{attribute 'qualified_only'}
{attribute 'strict'}
TYPE Motor :
(
	RotationMotor := 0,
	LiftingMotor := 1,
	ExtensionMotor := 2,
	GripMotor := 3
);
END_TYPE

(* stored: Version 1.1.0.1, ProductVersion 3.1.4024.13
   EnumerationTextList Motor: Id {e07e6d8d-4065-4147-a1dd-01b027a1ccda} *)
